// SIMATIC S7-200 project (STEP 7-Micro/WIN), CPU 222 REL 01.22

SYMBOL_TABLE USUARIO1
FR1              I0.0     // RELE TERMICO 1
FR2              I0.1     // RELE TERMICO 2
FR3              I0.2     // TELE TERMICO 3
S1               I0.3     // PULSADOR PARO
S2               I0.4     // PULSADOR MARCHA
KM1              Q0.0     // MOTOR 1
KM2              Q0.1     // MOTOR 2
KM3              Q0.2     // MOTOR 3
END_SYMBOL_TABLE

ORGANIZATION_BLOCK PRINCIPAL:OB1
TITLE=COMENTARIOS DEL PROGRAMA
BEGIN
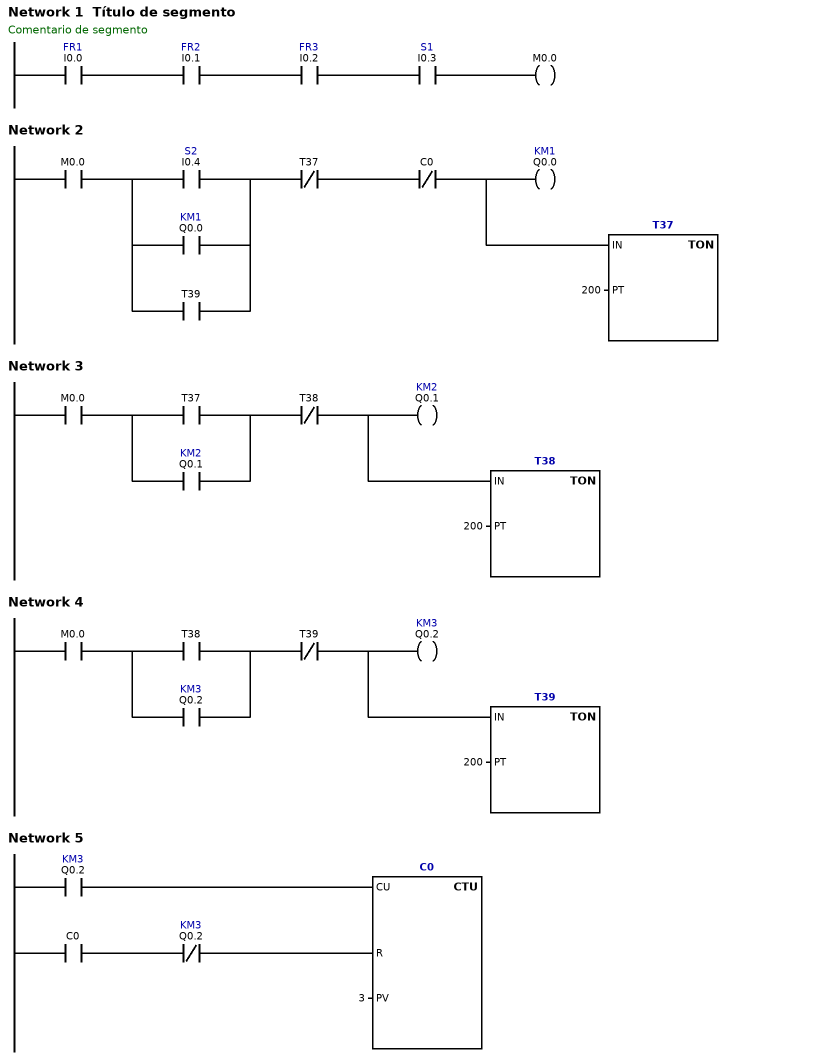
Network 1 // Título de segmento
// Comentario de segmento
LD     FR1:I0.0
A      FR2:I0.1
A      FR3:I0.2
A      S1:I0.3
=      M0.0
Network 2
LD     M0.0
LD     S2:I0.4
O      KM1:Q0.0
O      T39
ALD
AN     T37
AN     C0
=      KM1:Q0.0
TON    T37, 200
Network 3
LD     M0.0
LD     T37
O      KM2:Q0.1
ALD
AN     T38
=      KM2:Q0.1
TON    T38, 200
Network 4
LD     M0.0
LD     T38
O      KM3:Q0.2
ALD
AN     T39
=      KM3:Q0.2
TON    T39, 200
Network 5
LD     KM3:Q0.2
LD     C0
AN     KM3:Q0.2
CTU    C0, 3
END_ORGANIZATION_BLOCK
